ABB RobotStudio station: Fourth Assignment.rspag

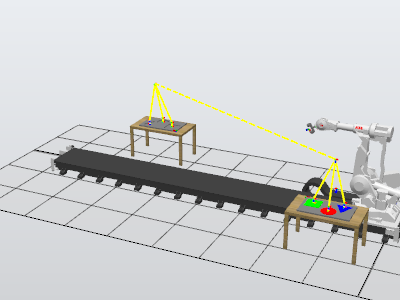
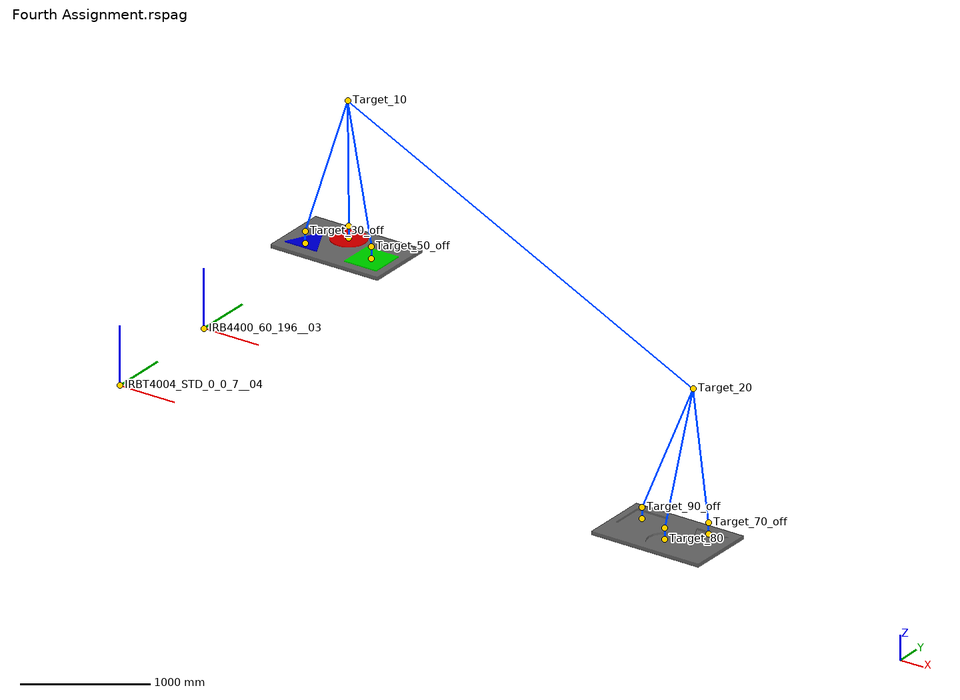
[picture v1: parts stored in the station drawn from their meshes, with robot base, taught points and paths (robot models come from the ABB library and are not in the file)]
--- station ---
Station Station (saved by RobotStudio 24.1.10713.1)
Controller Controller4, task T_ROB1: task frame (RAPID world) sits at (395.5, 560, 374.5) mm in the station
Controller Controller4
  mechanical unit ROB_1: IRB4400_60_196__03, 6 joints, base frame (0, 0, 0) mm
  mechanical unit TRACK_1: IRBT4004_STD_0_0_7__04, 1 joints, base frame (0, 0, 0) mm
Layout (positions relative to the parent item):
  - IRB4400_60_196__03 [mechanism, from %ABB.RobotStudio.Models.IRB4400%\IRB4400_60_196_G_03.rslib] at (395.5, 560, 374.5) mm; joint values [-0.5165, 0.1676, -0.1265, 0.0109, 1.138, -0.5864] (rad or m)
  - Table [part, from Move_parts\Table.rslib] at (1700, 1200, 0) mm
  - Table_2 [part, from Move_parts\Table.rslib] at (5200, -700, 0) mm, rotated rx 0 ry 0 rz 180 deg
  - IRBT4004_STD_0_0_7__04 [mechanism] at (0, 0, 0) mm; joint values [3.4756] (rad or m)
      links: Base, Link1
  - supportFrame [part] at (502.5, 1300, 828) mm, size 1000 x 600 x 30 mm
  - supportFrame_2 [part] at (6397.5, -800, 828) mm, rotated rx 0 ry 0 rz 180 deg, size 1000 x 600 x 30 mm
  - cirkel [part] at (502.5, 1300, 828) mm, size 300 x 298.4 x 30 mm
  - kvadrat [part] at (502.5, 1300, 828) mm, size 300 x 300 x 30 mm
  - triangel [part] at (502.5, 1300, 828) mm, size 300 x 300 x 30 mm
  - vacumtool [mechanism, from assignments 4\vacumtool.rslib] at (1596.74, 560, 2024.5) mm, rotated rx 180 ry 60 rz 180 deg
Attachment: IRB4400_60_196__03 is attached to IRBT4004_STD_0_0_7__04 / Link1
Attachment: vacumtool is attached to IRB4400_60_196__03 / Link6
EventTableEntry 4351: Group=, Trigger=DiOut 4352, Actions=[EventTableActionAttach 4353], Comment=, ActivationMode=2, Cyclic=false
EventTableTriggerIO 4352: IOValue=[1], IRC5Controller=? -1, Operator=0, SignalSource=Controller4 2450
EventTableActionAttach 4353: AttachmentParent=vacumtool 2444, AttachmentChild=? -1, MountObject=false, Offset=[X=1, Y=0, Z=0, W=0, X=0, Y=1, Z=0, W=0, X=0, Y=0, Z=1, W=0, X=0, Y=0, Z=0, W=1], FlangeIndext=0, FindNearest=true
EventTableEntry 4354: Group=, Trigger=DiOut 4355, Actions=[EventTableActionDetach 4356], Comment=, ActivationMode=2, Cyclic=false
EventTableTriggerIO 4355: IOValue=[0], IRC5Controller=? -1, Operator=0, SignalSource=Controller4 2450
EventTableActionDetach 4356: AttachmentParent=vacumtool 2444, AttachmentChild=? -1

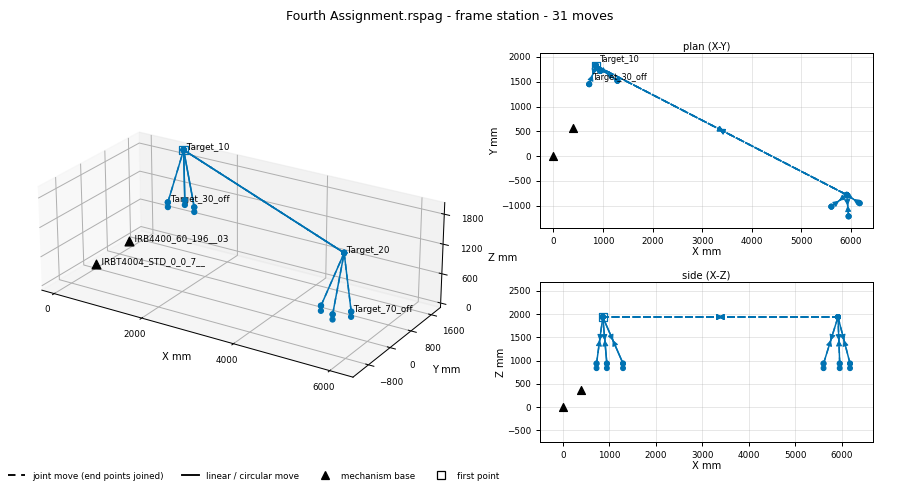
[picture p0: tool path of Fourth Assignment.rspag in frame station, 31 of 31 moves have a stored position in this frame; points joined in program order, loops and branches not executed]
--- Backups/Controller4/RAPID/TASK1/PROGMOD/CalibData.mod ---
MODULE CalibData
    PERS tooldata vacumtool:=[TRUE,[[0,0,170],[1,0,0,0]],[1,[0,0,1],[1,0,0,0],0,0,0]];
    TASK PERS wobjdata Workobject_1:=[FALSE,TRUE,"",[[1107,740,453.5],[0,0,1,0]],[[0,0,0],[1,0,0,0]]];
    TASK PERS wobjdata Workobject_2:=[FALSE,TRUE,"",[[5002,-1360,453.5],[0,1,0,0]],[[0,0,0],[1,0,0,0]]];
ENDMODULE

--- Backups/Controller4/RAPID/TASK1/PROGMOD/Module1.mod ---
MODULE Module1
    CONST robtarget Target_10:=[[645.796824836,527.145309545,-1111.499996088],[1,0,0,0],[0,0,0,0],[0,9E+09,9E+09,9E+09,9E+09,9E+09]];
    CONST robtarget Target_60:=[[684.130856077,405.684666035,-480.61684166],[0.156160962,0.052223292,-0.225734225,-0.960172142],[0,-1,-2,0],[0,9E+09,9E+09,9E+09,9E+09,9E+09]];
    CONST robtarget Target_30_off:=[[780,150,-110],[1,0,0,0],[0,0,0,0],[0,9E+09,9E+09,9E+09,9E+09,9E+09]];
    CONST robtarget Target_30:=[[780,150,-10],[1,0,0,0],[0,0,0,0],[0,9E+09,9E+09,9E+09,9E+09,9E+09]];
    CONST robtarget Target_20:=[[520.877935519,-18.474211931,-1111.499996088],[0.043938071,0.025367575,0.4,0.864910083],[-1,0,-2,0],[5386.224489796,9E+09,9E+09,9E+09,9E+09,9E+09]];
    CONST robtarget Target_40_off:=[[558.034,415.65,-110],[1,0,0,0],[0,0,0,0],[0,9E+09,9E+09,9E+09,9E+09,9E+09]];
    CONST robtarget Target_40:=[[558.034,415.65,-10],[1,0,0,0],[0,0,0,0],[0,9E+09,9E+09,9E+09,9E+09,9E+09]];
    CONST robtarget Target_50_off:=[[210,220,-110],[1,0,0,0],[0,0,0,0],[0,9E+09,9E+09,9E+09,9E+09,9E+09]];
    CONST robtarget Target_50:=[[210,220,-10],[1,0,0,0],[0,0,0,0],[0,9E+09,9E+09,9E+09,9E+09,9E+09]];
    CONST robtarget Target_70:=[[780,150,-10],[1,0,0,0],[-1,0,-3,0],[5386.224746704,9E+09,9E+09,9E+09,9E+09,9E+09]];
    CONST robtarget Target_70_off:=[[780,150,-110],[1,0,0,0],[-1,0,-3,0],[5386.224746704,9E+09,9E+09,9E+09,9E+09,9E+09]];
    CONST robtarget Target_80:=[[558.034,415.65,-10],[0,0,0,1],[-1,0,-1,0],[5386.224746704,9E+09,9E+09,9E+09,9E+09,9E+09]];
    CONST robtarget Target_80_off:=[[558.034,415.65,-110],[0,0,0,1],[-1,0,-1,0],[5386.224746704,9E+09,9E+09,9E+09,9E+09,9E+09]];
    CONST robtarget Target_90:=[[210,220,-10],[0,0,0,1],[-2,0,-2,0],[5386.224746704,9E+09,9E+09,9E+09,9E+09,9E+09]];
    CONST robtarget Target_90_off:=[[210,220,-110],[0,0,0,1],[-2,0,-2,0],[5386.224746704,9E+09,9E+09,9E+09,9E+09,9E+09]];

    PROC Path_10()
        MoveJ Target_10,v1000,fine,vacumtool\WObj:=Workobject_1;
        MoveL Target_30_off,v1000,fine,vacumtool\WObj:=Workobject_1;
        MoveL Target_30,v1000,fine,vacumtool\WObj:=Workobject_1;
        WaitTime 1;
        SetDO DiOut,1;
        WaitTime 1;
        MoveL Target_30_off,v1000,fine,vacumtool\WObj:=Workobject_1;
        MoveJ Target_10,v1000,fine,vacumtool\WObj:=Workobject_1;

        MoveJ Target_20,v1000,fine,vacumtool\WObj:=Workobject_2;
        MoveL Target_70_off,v1000,fine,vacumtool\WObj:=Workobject_2;
        MoveL Target_70,v1000,fine,vacumtool\WObj:=Workobject_2;
        WaitTime 1;
        SetDO DiOut,0;
        WaitTime 1;
        MoveL Target_70_off,v1000,fine,vacumtool\WObj:=Workobject_2;
        MoveJ Target_20,v1000,fine,vacumtool\WObj:=Workobject_2;

        MoveJ Target_10,v1000,fine,vacumtool\WObj:=Workobject_1;
        MoveL Target_40_off,v1000,fine,vacumtool\WObj:=Workobject_1;
        MoveL Target_40,v1000,fine,vacumtool\WObj:=Workobject_1;
        WaitTime 1;
        SetDO DiOut,1;
        WaitTime 1;
        MoveL Target_40_off,v1000,fine,vacumtool\WObj:=Workobject_1;
        MoveL Target_10,v1000,fine,vacumtool\WObj:=Workobject_1;

        MoveJ Target_20,v1000,fine,vacumtool\WObj:=Workobject_2;
        MoveL Target_80_off,v1000,fine,vacumtool\WObj:=Workobject_2;
        MoveL Target_80,v1000,fine,vacumtool\WObj:=Workobject_2;
        WaitTime 1;
        SetDO DiOut,0;
        WaitTime 1;
        MoveL Target_80_off,v1000,fine,vacumtool\WObj:=Workobject_2;
        MoveJ Target_20,v1000,fine,vacumtool\WObj:=Workobject_2;

        MoveJ Target_10,v1000,fine,vacumtool\WObj:=Workobject_1;
        MoveL Target_50_off,v1000,fine,vacumtool\WObj:=Workobject_1;
        MoveL Target_50,v1000,fine,vacumtool\WObj:=Workobject_1;
        WaitTime 1;
        SetDO DiOut,1;
        WaitTime 1;
        MoveL Target_50_off,v1000,fine,vacumtool\WObj:=Workobject_1;
        MoveL Target_10,v1000,fine,vacumtool\WObj:=Workobject_1;

        MoveJ Target_20,v1000,fine,vacumtool\WObj:=Workobject_2;
        MoveL Target_90_off,v1000,fine,vacumtool\WObj:=Workobject_2;
        MoveL Target_90,v1000,fine,vacumtool\WObj:=Workobject_2;
        WaitTime 1;
        SetDO DiOut,0;
        WaitTime 1;
        MoveL Target_90_off,v1000,fine,vacumtool\WObj:=Workobject_2;
        MoveJ Target_20,v1000,fine,vacumtool\WObj:=Workobject_2;

        MoveJ Target_10,v1000,fine,vacumtool\WObj:=Workobject_1;
    ENDPROC
    PROC main()
        SetDO DiOut,0;
        Path_10;
    ENDPROC
ENDMODULE

--- Backups/Controller4/SYSPAR/EIO.cfg ---
EIO:CFG_1.0:6:1::
#
INDUSTRIAL_NETWORK:

      -Name "PROFIBUS" -Label "PROFIBUS Controller Network"\
      -CfgPath "HOME/pbus_cfg.bin"
#
PROFIBUS_DEVICE:

      -Name "Board10"
#
EIO_SIGNAL:

      -Name "DiOut" -SignalType "DO" -Device "Board10" -DeviceMap "0"
